FUNCTION_BLOCK PUBLISH_OPCUA_4 (* Composite Function Block Type *)
  (* Standard: 61499-2 *)
  (* Version 1.0, 2019-02-09, iotdeveloperpk *)
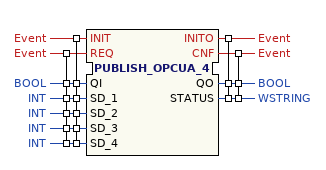
  EVENT_INPUT
    INIT WITH QI, SD_1, SD_2, SD_3, SD_4; (* Initialization Request *)
    REQ WITH QI, SD_1, SD_2, SD_3, SD_4; (* Normal Execution Request *)
  END_EVENT
  EVENT_OUTPUT
    INITO WITH QO, STATUS; (* Initialization Confirm *)
    CNF WITH QO, STATUS; (* Execution Confirmation *)
  END_EVENT
  VAR_INPUT
    QI : BOOL; (* Input event qualifier *)
    SD_1 : INT;
    SD_2 : INT;
    SD_3 : INT;
    SD_4 : INT;
  END_VAR
  VAR_OUTPUT
    QO : BOOL; (* Output event qualifier *)
    STATUS : WSTRING;
  END_VAR
  FBS
    PUBLISH_1 : PUBLISH_1(ID := opc_ua[/Objects/1:variables]);
    PUBLISH_1_1 : PUBLISH_1(ID := opc_ua[/Objects/2:variables]);
    PUBLISH_1_2 : PUBLISH_1(ID := opc_ua[/Objects/3:variables]);
    PUBLISH_1_3 : PUBLISH_1(ID := opc_ua[/Objects/4:variables]);
    variable1 : INT2INT;
    variable2 : INT2INT;
    variable3 : INT2INT;
    variable4 : INT2INT;
  END_FBS
  EVENT_CONNECTIONS
    INIT TO PUBLISH_1.INIT;
    INIT TO PUBLISH_1_1.INIT;
    INIT TO PUBLISH_1_2.INIT;
    INIT TO PUBLISH_1_3.INIT;
    PUBLISH_1.CNF TO CNF;
    REQ TO variable1.REQ;
    REQ TO variable2.REQ;
    REQ TO variable3.REQ;
    REQ TO variable4.REQ;
    variable4.CNF TO PUBLISH_1_3.REQ;
    variable3.CNF TO PUBLISH_1_2.REQ;
    variable2.CNF TO PUBLISH_1_1.REQ;
    variable1.CNF TO PUBLISH_1.REQ;
    PUBLISH_1.INITO TO INITO;
  END_CONNECTIONS
  DATA_CONNECTIONS
    QI TO PUBLISH_1.QI;
    QI TO PUBLISH_1_2.QI;
    QI TO PUBLISH_1_1.QI;
    QI TO PUBLISH_1_3.QI;
    PUBLISH_1.QO TO QO;
    variable1.OUT TO PUBLISH_1.SD_1;
    variable2.OUT TO PUBLISH_1_1.SD_1;
    variable3.OUT TO PUBLISH_1_2.SD_1;
    variable4.OUT TO PUBLISH_1_3.SD_1;
    PUBLISH_1.STATUS TO STATUS;
    SD_1 TO variable1.IN;
    SD_2 TO variable2.IN;
    SD_3 TO variable3.IN;
    SD_4 TO variable4.IN;
  END_CONNECTIONS
END_FUNCTION_BLOCK
